// TIA Portal V18 export
// export: Created 2026-01-09T11:32:10.2409871Z, ExportSetting WithDefaults, DisplayName Totally Integrated Automation Portal, DisplayVersion V18 Update 5, DisplayName TIA Portal Openness, DisplayVersion V18 Update 5, DisplayName TIA Portal Teamcenter Gateway, DisplayVersion V18, DisplayName TIA Portal Version Control Interface, DisplayVersion V18, DisplayName SINAMICS Startdrive Advanced, DisplayVersion V18 SP2 Update 1, DisplayName SINAMICS Startdrive G110M, G120, G120C, G120D, G120P, G115D, DisplayVersion V18 SP2 Update 1, DisplayName SINAMICS Startdrive G130, G150, S120, S150, SINAMICS MV, S210, G220, S200, DisplayVersion V18 SP2 Update 1, DisplayName STEP 7 Professional, DisplayVersion V18 Update 5, DisplayName STEP 7 Safety, DisplayVersion V18, DisplayName WinCC Professional, DisplayVersion V18 Update 5
TagTable "Presser"
  KistlerPresser_ContinueSeq : Bool  (%DB[KistlerPresser_DB_Number].DBX110.4, CPU S71500-2PN_TP700, 100 ms)
  KistlerPresser_Homing : Bool  (%DB[KistlerPresser_DB_Number].DBX110.2, CPU S71500-2PN_TP700, 100 ms)
  KistlerPresser_Inputs_ACK : Bool  (%DB[KistlerPresser_DB_Number].DBX199.1, CPU S71500-2PN_TP700, 100 ms)
  KistlerPresser_Inputs_ALARM : Bool  (%DB[KistlerPresser_DB_Number].DBX186.7, CPU S71500-2PN_TP700, 100 ms)
  KistlerPresser_Inputs_AUTO : Bool  (%DB[KistlerPresser_DB_Number].DBX181.4, CPU S71500-2PN_TP700, 100 ms)
  KistlerPresser_Inputs_BACKUP-REQUEST : Bool  (%DB[KistlerPresser_DB_Number].DBX199.7, CPU S71500-2PN_TP700, 100 ms)
  KistlerPresser_Inputs_BRAKETEST-DONE : Bool  (%DB[KistlerPresser_DB_Number].DBX189.7, CPU S71500-2PN_TP700, 100 ms)
  KistlerPresser_Inputs_BRAKETEST-REQ : Bool  (%DB[KistlerPresser_DB_Number].DBX191.1, CPU S71500-2PN_TP700, 100 ms)
  KistlerPresser_Inputs_BREAKETEST-ACTIVE : Bool  (%DB[KistlerPresser_DB_Number].DBX183.5, CPU S71500-2PN_TP700, 100 ms)
  KistlerPresser_Inputs_CFG-MP : Byte  (%DB[KistlerPresser_DB_Number].DBB194, CPU S71500-2PN_TP700, 100 ms)
  KistlerPresser_Inputs_CHANGED--GLOBAL : Bool  (%DB[KistlerPresser_DB_Number].DBX199.6, CPU S71500-2PN_TP700, 100 ms)
  KistlerPresser_Inputs_CHANGEDSELECTED-MP : Bool  (%DB[KistlerPresser_DB_Number].DBX199.4, CPU S71500-2PN_TP700, 100 ms)
  KistlerPresser_Inputs_DEVICE-AVAILABLE : Bool  (%DB[KistlerPresser_DB_Number].DBX199.2, CPU S71500-2PN_TP700, 100 ms)
  KistlerPresser_Inputs_DRIVE-ENABLE : Bool  (%DB[KistlerPresser_DB_Number].DBX189.0, CPU S71500-2PN_TP700, 100 ms)
  KistlerPresser_Inputs_DRIVE-ENABLED : Bool  (%DB[KistlerPresser_DB_Number].DBX190.5, CPU S71500-2PN_TP700, 100 ms)
  KistlerPresser_Inputs_DRIVE-TO-HOMEPOS : Bool  (%DB[KistlerPresser_DB_Number].DBX189.2, CPU S71500-2PN_TP700, 100 ms)
  KistlerPresser_Inputs_DRIVE-TO-REFPOS : Bool  (%DB[KistlerPresser_DB_Number].DBX189.3, CPU S71500-2PN_TP700, 100 ms)
  KistlerPresser_Inputs_EXT-STOP : Bool  (%DB[KistlerPresser_DB_Number].DBX190.3, CPU S71500-2PN_TP700, 100 ms)
  KistlerPresser_Inputs_GLOBAL-CFG-MP : Bool  (%DB[KistlerPresser_DB_Number].DBX195.7, CPU S71500-2PN_TP700, 100 ms)
  KistlerPresser_Inputs_HOMEPOS-REACHED : Bool  (%DB[KistlerPresser_DB_Number].DBX190.6, CPU S71500-2PN_TP700, 100 ms)
  KistlerPresser_Inputs_INC-ZERO : Bool  (%DB[KistlerPresser_DB_Number].DBX180.7, CPU S71500-2PN_TP700, 100 ms)
  KistlerPresser_Inputs_JOG-BW : Bool  (%DB[KistlerPresser_DB_Number].DBX189.5, CPU S71500-2PN_TP700, 100 ms)
  KistlerPresser_Inputs_JOG-FW : Bool  (%DB[KistlerPresser_DB_Number].DBX189.4, CPU S71500-2PN_TP700, 100 ms)
  KistlerPresser_Inputs_LABEL-ID : Byte  (%DB[KistlerPresser_DB_Number].DBB193, CPU S71500-2PN_TP700, 100 ms)
  KistlerPresser_Inputs_MASTER-MEAS : Bool  (%DB[KistlerPresser_DB_Number].DBX180.6, CPU S71500-2PN_TP700, 100 ms)
  KistlerPresser_Inputs_MIRRIR-CFG-ADR : Byte  (%DB[KistlerPresser_DB_Number].DBB196, CPU S71500-2PN_TP700, 100 ms)
  KistlerPresser_Inputs_MIRRIR-CFG-LENGTH : Byte  (%DB[KistlerPresser_DB_Number].DBB197, CPU S71500-2PN_TP700, 100 ms)
  KistlerPresser_Inputs_MIRROR-ACCESS : Bool  (%DB[KistlerPresser_DB_Number].DBX181.3, CPU S71500-2PN_TP700, 100 ms)
  KistlerPresser_Inputs_MIRROR-ACK-ADMIN : Bool  (%DB[KistlerPresser_DB_Number].DBX181.1, CPU S71500-2PN_TP700, 100 ms)
  KistlerPresser_Inputs_MIRROR-START : Bool  (%DB[KistlerPresser_DB_Number].DBX180.0, CPU S71500-2PN_TP700, 100 ms)
  KistlerPresser_Inputs_MIRROR-STEST-X : Bool  (%DB[KistlerPresser_DB_Number].DBX180.3, CPU S71500-2PN_TP700, 100 ms)
  KistlerPresser_Inputs_MIRROR-STEST-Y : Bool  (%DB[KistlerPresser_DB_Number].DBX180.4, CPU S71500-2PN_TP700, 100 ms)
  KistlerPresser_Inputs_MIRROR-TARE-Y : Bool  (%DB[KistlerPresser_DB_Number].DBX180.1, CPU S71500-2PN_TP700, 100 ms)
  KistlerPresser_Inputs_MIRROR-ZERO X : Bool  (%DB[KistlerPresser_DB_Number].DBX180.2, CPU S71500-2PN_TP700, 100 ms)
  KistlerPresser_Inputs_MP : Byte  (%DB[KistlerPresser_DB_Number].DBB182, CPU S71500-2PN_TP700, 100 ms)
  KistlerPresser_Inputs_NOK-TOTAL : Bool  (%DB[KistlerPresser_DB_Number].DBX186.2, CPU S71500-2PN_TP700, 100 ms)
  KistlerPresser_Inputs_NO-PASS : Bool  (%DB[KistlerPresser_DB_Number].DBX186.3, CPU S71500-2PN_TP700, 100 ms)
  KistlerPresser_Inputs_OK-TOTAL : Bool  (%DB[KistlerPresser_DB_Number].DBX186.1, CPU S71500-2PN_TP700, 100 ms)
  KistlerPresser_Inputs_ONLINE-EO-NOK : Bool  (%DB[KistlerPresser_DB_Number].DBX190.2, CPU S71500-2PN_TP700, 100 ms)
  KistlerPresser_Inputs_READY : Bool  (%DB[KistlerPresser_DB_Number].DBX186.0, CPU S71500-2PN_TP700, 100 ms)
  KistlerPresser_Inputs_REFPOS-REACHED : Bool  (%DB[KistlerPresser_DB_Number].DBX190.7, CPU S71500-2PN_TP700, 100 ms)
  KistlerPresser_Inputs_RESET-SN-GENERATOR : Bool  (%DB[KistlerPresser_DB_Number].DBX183.2, CPU S71500-2PN_TP700, 100 ms)
  KistlerPresser_Inputs_RUN-SEQUENCE : Bool  (%DB[KistlerPresser_DB_Number].DBX189.1, CPU S71500-2PN_TP700, 100 ms)
  KistlerPresser_Inputs_S1 : Bool  (%DB[KistlerPresser_DB_Number].DBX187.0, CPU S71500-2PN_TP700, 100 ms)
  KistlerPresser_Inputs_S2 : Bool  (%DB[KistlerPresser_DB_Number].DBX187.1, CPU S71500-2PN_TP700, 100 ms)
  KistlerPresser_Inputs_SELECT-PAGE : Byte  (%DB[KistlerPresser_DB_Number].DBB198, CPU S71500-2PN_TP700, 100 ms)
  KistlerPresser_Inputs_SEQUENCE : Byte  (%DB[KistlerPresser_DB_Number].DBB192, CPU S71500-2PN_TP700, 100 ms)
  KistlerPresser_Inputs_SEQUENCE-END : Bool  (%DB[KistlerPresser_DB_Number].DBX190.1, CPU S71500-2PN_TP700, 100 ms)
  KistlerPresser_Inputs_SEQUENCE-ERROR : Bool  (%DB[KistlerPresser_DB_Number].DBX190.4, CPU S71500-2PN_TP700, 100 ms)
  KistlerPresser_Inputs_SEQUENCE-STOPPED : Bool  (%DB[KistlerPresser_DB_Number].DBX190.0, CPU S71500-2PN_TP700, 100 ms)
  KistlerPresser_Inputs_SERVO-ERROR : Bool  (%DB[KistlerPresser_DB_Number].DBX191.3, CPU S71500-2PN_TP700, 100 ms)
  KistlerPresser_Inputs_SERVO-WARN : Bool  (%DB[KistlerPresser_DB_Number].DBX191.2, CPU S71500-2PN_TP700, 100 ms)
  KistlerPresser_Inputs_SMES-ACTIVE : Bool  (%DB[KistlerPresser_DB_Number].DBX191.4, CPU S71500-2PN_TP700, 100 ms)
  KistlerPresser_Inputs_SMM1-ACTIVE : Bool  (%DB[KistlerPresser_DB_Number].DBX191.6, CPU S71500-2PN_TP700, 100 ms)
  KistlerPresser_Inputs_SMST2-ACTIVE : Bool  (%DB[KistlerPresser_DB_Number].DBX191.5, CPU S71500-2PN_TP700, 100 ms)
  KistlerPresser_Inputs_STANDSTILL : Bool  (%DB[KistlerPresser_DB_Number].DBX191.0, CPU S71500-2PN_TP700, 100 ms)
  KistlerPresser_Inputs_STAT-DISABLE : Bool  (%DB[KistlerPresser_DB_Number].DBX181.6, CPU S71500-2PN_TP700, 100 ms)
  KistlerPresser_Inputs_STAT-RESET : Bool  (%DB[KistlerPresser_DB_Number].DBX181.5, CPU S71500-2PN_TP700, 100 ms)
  KistlerPresser_Inputs_TARE-EXTENDED-Y : Bool  (%DB[KistlerPresser_DB_Number].DBX181.7, CPU S71500-2PN_TP700, 100 ms)
  KistlerPresser_Inputs_TRANSMISSION-FAULT : Bool  (%DB[KistlerPresser_DB_Number].DBX199.0, CPU S71500-2PN_TP700, 100 ms)
  KistlerPresser_Inputs_USER-MODE-ACTIVE : Bool  (%DB[KistlerPresser_DB_Number].DBX191.7, CPU S71500-2PN_TP700, 100 ms)
  KistlerPresser_Inputs_WAIT-REQUEST : Bool  (%DB[KistlerPresser_DB_Number].DBX189.6, CPU S71500-2PN_TP700, 100 ms)
  KistlerPresser_Inputs_WARN : Bool  (%DB[KistlerPresser_DB_Number].DBX186.6, CPU S71500-2PN_TP700, 100 ms)
  KistlerPresser_JogNeg : Bool  (%DB[KistlerPresser_DB_Number].DBX110.6, CPU S71500-2PN_TP700, 100 ms)
  KistlerPresser_JogPos : Bool  (%DB[KistlerPresser_DB_Number].DBX110.5, CPU S71500-2PN_TP700, 100 ms)
  KistlerPresser_Outputs_ACCESS : Bool  (%DB[KistlerPresser_DB_Number].DBX401.3, CPU S71500-2PN_TP700, 100 ms)
  KistlerPresser_Outputs_ACK-ADMIN : Bool  (%DB[KistlerPresser_DB_Number].DBX401.1, CPU S71500-2PN_TP700, 100 ms)
  KistlerPresser_Outputs_AUTO : Bool  (%DB[KistlerPresser_DB_Number].DBX401.4, CPU S71500-2PN_TP700, 100 ms)
  KistlerPresser_Outputs_BACKUP-REQUEST : Bool  (%DB[KistlerPresser_DB_Number].DBX419.7, CPU S71500-2PN_TP700, 100 ms)
  KistlerPresser_Outputs_CONTNUEFROM-WAIT : Bool  (%DB[KistlerPresser_DB_Number].DBX409.6, CPU S71500-2PN_TP700, 100 ms)
  KistlerPresser_Outputs_DRIVE-ENABLE : Bool  (%DB[KistlerPresser_DB_Number].DBX409.0, CPU S71500-2PN_TP700, 100 ms)
  KistlerPresser_Outputs_DRIVE-TO-HOMEPOS : Bool  (%DB[KistlerPresser_DB_Number].DBX409.2, CPU S71500-2PN_TP700, 100 ms)
  KistlerPresser_Outputs_DRIVE-TO-REFPOS : Bool  (%DB[KistlerPresser_DB_Number].DBX409.3, CPU S71500-2PN_TP700, 100 ms)
  KistlerPresser_Outputs_GLOBAL-CFG-MP : Bool  (%DB[KistlerPresser_DB_Number].DBX415.7, CPU S71500-2PN_TP700, 100 ms)
  KistlerPresser_Outputs_INC-ZERO : Bool  (%DB[KistlerPresser_DB_Number].DBX400.7, CPU S71500-2PN_TP700, 100 ms)
  KistlerPresser_Outputs_JOG-BW : Bool  (%DB[KistlerPresser_DB_Number].DBX409.5, CPU S71500-2PN_TP700, 100 ms)
  KistlerPresser_Outputs_JOG-FW : Bool  (%DB[KistlerPresser_DB_Number].DBX409.4, CPU S71500-2PN_TP700, 100 ms)
  KistlerPresser_Outputs_MANUAL-BRAKETEST : Bool  (%DB[KistlerPresser_DB_Number].DBX409.7, CPU S71500-2PN_TP700, 100 ms)
  KistlerPresser_Outputs_MASTER-MEAS : Bool  (%DB[KistlerPresser_DB_Number].DBX400.6, CPU S71500-2PN_TP700, 100 ms)
  KistlerPresser_Outputs_RESET-CHANGEDGLOBAL : Bool  (%DB[KistlerPresser_DB_Number].DBX419.6, CPU S71500-2PN_TP700, 100 ms)
  KistlerPresser_Outputs_RESET-CHANGED-SELECTED-MP : Bool  (%DB[KistlerPresser_DB_Number].DBX419.4, CPU S71500-2PN_TP700, 100 ms)
  KistlerPresser_Outputs_RESET-SN-GENERATOR : Bool  (%DB[KistlerPresser_DB_Number].DBX403.2, CPU S71500-2PN_TP700, 100 ms)
  KistlerPresser_Outputs_RUN-SEQUENCE : Bool  (%DB[KistlerPresser_DB_Number].DBX409.1, CPU S71500-2PN_TP700, 100 ms)
  KistlerPresser_Outputs_SAVE-TO-MP : Bool  (%DB[KistlerPresser_DB_Number].DBX419.0, CPU S71500-2PN_TP700, 100 ms)
  KistlerPresser_Outputs_SEQ-EXT-STOP-REQ : Bool  (%DB[KistlerPresser_DB_Number].DBX410.3, CPU S71500-2PN_TP700, 100 ms)
  KistlerPresser_Outputs_START : Bool  (%DB[KistlerPresser_DB_Number].DBX400.0, CPU S71500-2PN_TP700, 100 ms)
  KistlerPresser_Outputs_STAT-DISABLE : Bool  (%DB[KistlerPresser_DB_Number].DBX401.6, CPU S71500-2PN_TP700, 100 ms)
  KistlerPresser_Outputs_STAT-RESET : Bool  (%DB[KistlerPresser_DB_Number].DBX401.5, CPU S71500-2PN_TP700, 100 ms)
  KistlerPresser_Outputs_STEST-X : Bool  (%DB[KistlerPresser_DB_Number].DBX400.3, CPU S71500-2PN_TP700, 100 ms)
  KistlerPresser_Outputs_STEST-Y : Bool  (%DB[KistlerPresser_DB_Number].DBX400.4, CPU S71500-2PN_TP700, 100 ms)
  KistlerPresser_Outputs_STROBE : Bool  (%DB[KistlerPresser_DB_Number].DBX419.1, CPU S71500-2PN_TP700, 100 ms)
  KistlerPresser_Outputs_TARE-EXTENDED-Y : Bool  (%DB[KistlerPresser_DB_Number].DBX401.7, CPU S71500-2PN_TP700, 100 ms)
  KistlerPresser_Outputs_TARE-Y : Bool  (%DB[KistlerPresser_DB_Number].DBX400.1, CPU S71500-2PN_TP700, 100 ms)
  KistlerPresser_Outputs_ZERO X : Bool  (%DB[KistlerPresser_DB_Number].DBX400.2, CPU S71500-2PN_TP700, 100 ms)
  KistlerPresser_StartCycle : Bool  (%DB[KistlerPresser_DB_Number].DBX110.3, CPU S71500-2PN_TP700, 100 ms)
  KistlerPresser_DB_Number : Int  (100 ms)
  KistlerPresser_Inputs_FreelyConfigurableArea_CurValueX_1 : Real  (%DB[KistlerPresser_DB_Number].DBD204, CPU S71500-2PN_TP700, 100 ms)
  KistlerPresser_Inputs_FreelyConfigurableArea_CurValueY : Real  (%DB[KistlerPresser_DB_Number].DBD212, CPU S71500-2PN_TP700, 100 ms)
  KistlerPresser_oFltNo : Word  (%DB[KistlerPresser_DB_Number].DBW82, CPU S71500-2PN_TP700, 100 ms)
  KistlerPresser_Outputs_CFG-ADDRESS : Byte  (%DB[KistlerPresser_DB_Number].DBB416, CPU S71500-2PN_TP700, 100 ms)
  KistlerPresser_Outputs_CFG-LENGTH : Byte  (%DB[KistlerPresser_DB_Number].DBB417, CPU S71500-2PN_TP700, 100 ms)
  KistlerPresser_Outputs_CFG-MP : Byte  (%DB[KistlerPresser_DB_Number].DBB414, CPU S71500-2PN_TP700, 100 ms)
  KistlerPresser_Outputs_CURRENT SEQUENCE : Byte  (%DB[KistlerPresser_DB_Number].DBB412, CPU S71500-2PN_TP700, 100 ms)
  KistlerPresser_Outputs_FreelyConfigurableArea_JogMaxForce : Real  (%DB[KistlerPresser_DB_Number].DBD428, CPU S71500-2PN_TP700, 100 ms)
  KistlerPresser_Outputs_FreelyConfigurableArea_JogSpeed : Real  (%DB[KistlerPresser_DB_Number].DBD424, CPU S71500-2PN_TP700, 100 ms)
  KistlerPresser_Outputs_SELECT-PAGE : Byte  (%DB[KistlerPresser_DB_Number].DBB418, CPU S71500-2PN_TP700, 100 ms)
  KistlerPresser_ProgNo : Int  (%DB[KistlerPresser_DB_Number].DBW106, CPU S71500-2PN_TP700, 100 ms)
  KistlerPresser_SelectSeq : Int  (%DB[KistlerPresser_DB_Number].DBW108, CPU S71500-2PN_TP700, 100 ms)
  ProcessData_1_PressInterlock_1 : Array [0..15] of Bool  (PLC tag ProcessData_1.PressInterlock_1, CPU S71500-2PN_TP700, 1 s)
    TagArrayMember "[0]"
    TagArrayMember "[1]"
    TagArrayMember "[2]"
    TagArrayMember "[3]"
    TagArrayMember "[4]"
    TagArrayMember "[5]"
    TagArrayMember "[6]"
    TagArrayMember "[7]"
    TagArrayMember "[8]"
    TagArrayMember "[9]"
    TagArrayMember "[10]"
    TagArrayMember "[11]"
    TagArrayMember "[12]"
    TagArrayMember "[13]"
    TagArrayMember "[14]"
    TagArrayMember "[15]"
  ProcessData_1_PressInterlock_2 : Array [0..15] of Bool  (PLC tag ProcessData_1.PressInterlock_2, CPU S71500-2PN_TP700, 1 s)
    TagArrayMember "[0]"
    TagArrayMember "[1]"
    TagArrayMember "[2]"
    TagArrayMember "[3]"
    TagArrayMember "[4]"
    TagArrayMember "[5]"
    TagArrayMember "[6]"
    TagArrayMember "[7]"
    TagArrayMember "[8]"
    TagArrayMember "[9]"
    TagArrayMember "[10]"
    TagArrayMember "[11]"
    TagArrayMember "[12]"
    TagArrayMember "[13]"
    TagArrayMember "[14]"
    TagArrayMember "[15]"
  KistlerPressData2_ManualPro : Int  (PLC tag KistlerPressData2.ManualPro, CPU S71500-2PN_TP700, 1 s)
  KistlerPressData1_ManualPro : Int  (PLC tag KistlerPressData1.ManualPro, CPU S71500-2PN_TP700, 1 s)
  ProcessData_1_Calibartion_1 : Bool  (PLC tag ProcessData_1.Calibartion_1, CPU S71500-2PN_TP700, 1 s)
  ProcessData_1_Calibartion_2 : Bool  (PLC tag ProcessData_1.Calibartion_2, CPU S71500-2PN_TP700, 1 s)
